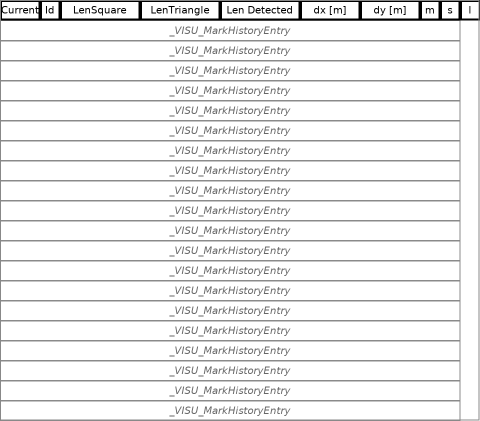
VISUALIZATION _VISU_MarkHistory  // 480x421
VAR_IN_OUT
	mInst : FB_MarkDetection;
END_VAR
    Frame (0,20 460x21)
        shows _VISU_MarkHistoryEntry(mInst := mInst.sMarkHistory[0])
    Rectangle (0,0 40x20), "Current"
    Rectangle (40,0 20x20), "Id"
    Rectangle (60,0 80x20), "LenSquare"
    Rectangle (140,0 80x20), "LenTriangle"
    Rectangle (220,0 80x20), "Len Detected"
    Rectangle (300,0 60x20), "dx [m]"
    Frame (0,40 460x21)
        shows _VISU_MarkHistoryEntry(mInst := mInst.sMarkHistory[1])
    Frame (0,60 460x21)
        shows _VISU_MarkHistoryEntry(mInst := mInst.sMarkHistory[2])
    Frame (0,80 460x21)
        shows _VISU_MarkHistoryEntry(mInst := mInst.sMarkHistory[3])
    Frame (0,100 460x21)
        shows _VISU_MarkHistoryEntry(mInst := mInst.sMarkHistory[4])
    Frame (0,120 460x21)
        shows _VISU_MarkHistoryEntry(mInst := mInst.sMarkHistory[5])
    Frame (0,140 460x21)
        shows _VISU_MarkHistoryEntry(mInst := mInst.sMarkHistory[6])
    Frame (0,160 460x21)
        shows _VISU_MarkHistoryEntry(mInst := mInst.sMarkHistory[7])
    Frame (0,180 460x21)
        shows _VISU_MarkHistoryEntry(mInst := mInst.sMarkHistory[8])
    Frame (0,200 460x21)
        shows _VISU_MarkHistoryEntry(mInst := mInst.sMarkHistory[9])
    Frame (0,220 460x21)
        shows _VISU_MarkHistoryEntry(mInst := mInst.sMarkHistory[10])
    Frame (0,240 460x21)
        shows _VISU_MarkHistoryEntry(mInst := mInst.sMarkHistory[11])
    Frame (0,260 460x21)
        shows _VISU_MarkHistoryEntry(mInst := mInst.sMarkHistory[12])
    Frame (0,280 460x21)
        shows _VISU_MarkHistoryEntry(mInst := mInst.sMarkHistory[13])
    Frame (0,300 460x21)
        shows _VISU_MarkHistoryEntry(mInst := mInst.sMarkHistory[14])
    Frame (0,320 460x21)
        shows _VISU_MarkHistoryEntry(mInst := mInst.sMarkHistory[15])
    Frame (0,340 460x21)
        shows _VISU_MarkHistoryEntry(mInst := mInst.sMarkHistory[16])
    Frame (0,360 460x21)
        shows _VISU_MarkHistoryEntry(mInst := mInst.sMarkHistory[17])
    Frame (0,380 460x21)
        shows _VISU_MarkHistoryEntry(mInst := mInst.sMarkHistory[18])
    Frame (0,400 460x21)
        shows _VISU_MarkHistoryEntry(mInst := mInst.sMarkHistory[19])
    Rectangle (360,0 60x20), "dy [m]"
    Rectangle (420,0 20x20), "m", tooltip "missed"
    Rectangle (440,0 20x20), "s", tooltip "too short"
    Rectangle (460,0 20x20), "l", tooltip "too long"
END_VISUALIZATION

(* stored: Version 1.1.0.1, ProductVersion 3.1.4024.11
   Visu _VISU_MarkHistory: Id {f153da49-d3a5-477b-b608-e86936198962} *)
